// TIA Portal V20 export
FUNCTION_BLOCK "CC_Main"   // FB100, LAD
{ S7_Optimized_Access := 'TRUE' }
// stored: AutoNumber false, MemoryReserve 100, SetENOAutomatically false
   VAR_INPUT
      HMI_Reset : Bool;
      ST23_Selected : Bool;
      CNT_DownPos1 : Bool;
      CNT_DownPos2 : Bool;
      CNT_UpPos1 : Bool;
      CNT_UpPos2 : Bool;
      Hydraulic_Roller_DownPos1 : Bool;
      Hydraulic_Roller_DownPos2 : Bool;
      Hydraulic_Roller_UpPos1 : Bool;
      Hydraulic_Roller_UpPos2 : Bool;
      Drive_Roller_DownPos1 : Bool;
      Drive_Roller_DownPos2 : Bool;
      Drive_Roller_UpPos1 : Bool;
      Drive_Roller_UpPos2 : Bool;
      Module_DownPos1 : Bool;
      Module_DownPos2 : Bool;
      Module_UpPos1 : Bool;
      Module_UpPos2 : Bool;
   END_VAR
   VAR_OUTPUT
      Hydraulic_Main_Valve_Control : Bool;
   END_VAR
   VAR
      Hydraulic_Unit_Active : Bool;
      Any_Valve_Active : Bool;
      HydUnitTimerOff { S7_SetPoint := 'True'} : TON_TIME;
      HydraulicUnit_MC_Power { S7_SetPoint := 'True'} : MC_POWER;
      HydraulicUnit_MC_MoveJog { S7_SetPoint := 'True'} : MC_MOVEJOG;
      HydraulicUnit_MC_Reset { S7_SetPoint := 'True'} : MC_RESET;
      Vibrator_Control_MOD1 { S7_SetPoint := 'True'} : "CC_Vibrator_Control";
      Vibrator_Control_MOD2 { S7_SetPoint := 'True'} : "CC_Vibrator_Control";
      Vibrator_Control_MOD3 { S7_SetPoint := 'True'} : "CC_Vibrator_Control";
      Module_Control_ST23 { S7_SetPoint := 'True'} : "CC_Vib_Modules";
      ST23_UP_whenMoving { S7_SetPoint := 'True'} : Bool;
      ST24_UP_whenMoving : Bool;
      ST25_UP_whenMoving : Bool;
      MC_Power_Vib1 { S7_SetPoint := 'True'} : MC_POWER;
      MC_RESET_Vib1 { S7_SetPoint := 'True'} : MC_RESET;
      MC_MOVEJOG_Vib1 { S7_SetPoint := 'True'} : MC_MOVEJOG;
      ST24_DriveRollsUP { S7_SetPoint := 'True'} : Bool;
      ST24_DriveRollsDown : Bool;
      ST25_DriveRollsUp : Bool;
      ST25_DriveRollsDown : Bool;
      ST23_Station_Control { S7_SetPoint := 'True'} : "CC_Station_Control";
      ST24_Station_Control { S7_SetPoint := 'True'} : "CC_Station_Control";
      ST25_Station_Control { S7_SetPoint := 'True'} : "CC_Station_Control";
      ST24_Selected : Bool;
   END_VAR
   VAR CONSTANT
      STEP_RETRACT : Int := 1;
      STEP_MOVING : Int := 2;
      STEP_EXTEND : Int := 3;
   END_VAR
BEGIN

REGION Network 1
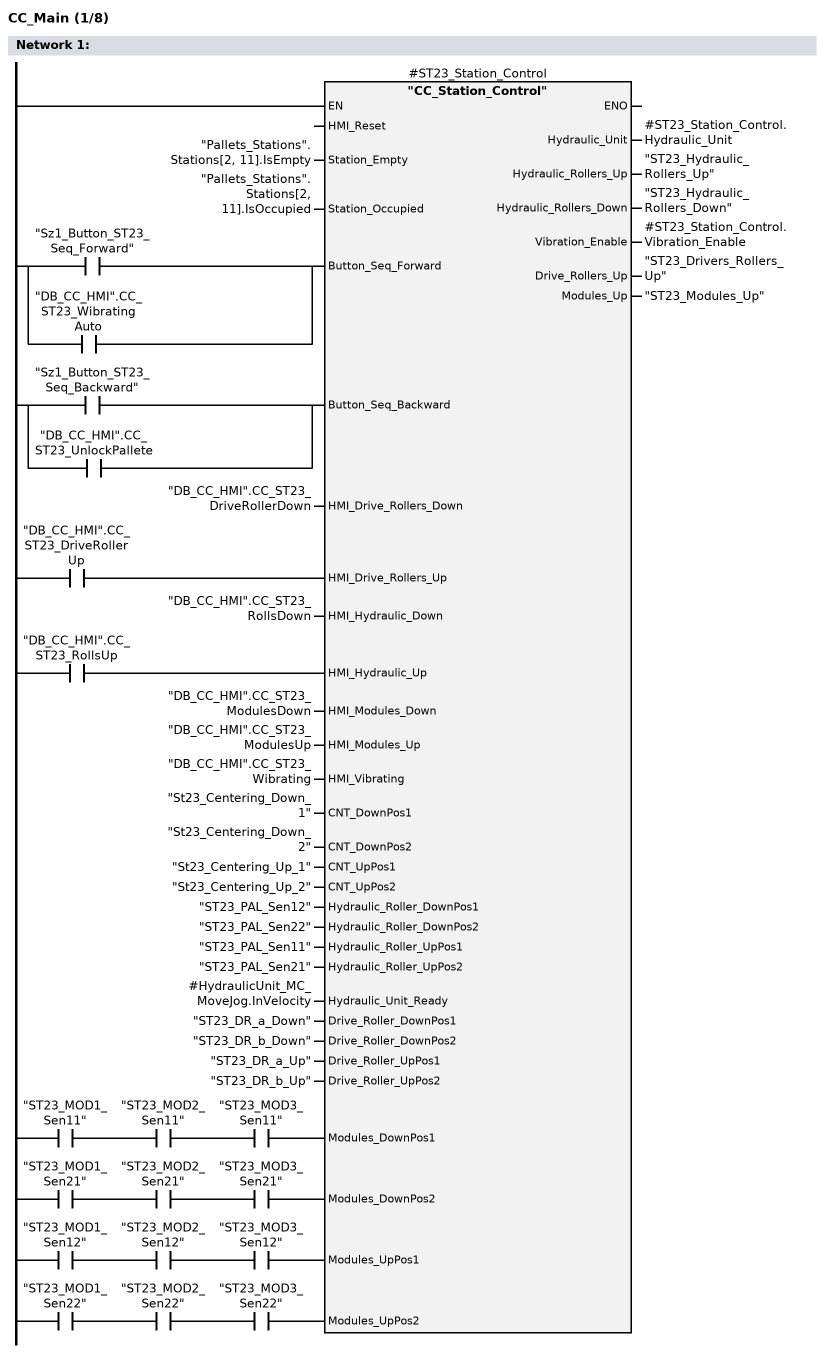
   RUNG wire#powerrail
      #ST23_Station_Control(Button_Seq_Forward := wire#w1, Button_Seq_Backward := wire#w2, HMI_Drive_Rollers_Up := wire#w3, HMI_Hydraulic_Up := wire#w4, Modules_DownPos1 := wire#w5, Modules_DownPos2 := wire#w6, Modules_UpPos1 := wire#w7, Modules_UpPos2 := wire#w8, HMI_Reset :=, Station_Empty := "Pallets_Stations".Stations[2, 11].IsEmpty, Station_Occupied := "Pallets_Stations".Stations[2, 11].IsOccupied, HMI_Drive_Rollers_Down := "DB_CC_HMI".CC_ST23_DriveRollerDown, HMI_Hydraulic_Down := "DB_CC_HMI".CC_ST23_RollsDown, HMI_Modules_Down := "DB_CC_HMI".CC_ST23_ModulesDown, HMI_Modules_Up := "DB_CC_HMI".CC_ST23_ModulesUp, HMI_Vibrating := "DB_CC_HMI".CC_ST23_Wibrating, CNT_DownPos1 := "St23_Centering_Down_1", CNT_DownPos2 := "St23_Centering_Down_2", CNT_UpPos1 := "St23_Centering_Up_1", CNT_UpPos2 := "St23_Centering_Up_2", Hydraulic_Roller_DownPos1 := "ST23_PAL_Sen12", Hydraulic_Roller_DownPos2 := "ST23_PAL_Sen22", Hydraulic_Roller_UpPos1 := "ST23_PAL_Sen11", Hydraulic_Roller_UpPos2 := "ST23_PAL_Sen21", Hydraulic_Unit_Ready := #HydraulicUnit_MC_MoveJog.InVelocity, Drive_Roller_DownPos1 := "ST23_DR_a_Down", Drive_Roller_DownPos2 := "ST23_DR_b_Down", Drive_Roller_UpPos1 := "ST23_DR_a_Up", Drive_Roller_UpPos2 := "ST23_DR_b_Up", Hydraulic_Unit => #ST23_Station_Control.Hydraulic_Unit, Hydraulic_Rollers_Up => "ST23_Hydraulic_Rollers_Up", Hydraulic_Rollers_Down => "ST23_Hydraulic_Rollers_Down", Vibration_Enable => #ST23_Station_Control.Vibration_Enable, Drive_Rollers_Up => "ST23_Drivers_Rollers_Up", Modules_Up => "ST23_Modules_Up")
   END_RUNG
   RUNG wire#powerrail
      Contact( "Sz1_Button_ST23_Seq_Forward" )
   END_RUNG wire#w1
   RUNG wire#powerrail
      Contact( "DB_CC_HMI".CC_ST23_WibratingAuto )
   END_RUNG wire#w1
   RUNG wire#powerrail
      Contact( "Sz1_Button_ST23_Seq_Backward" )
   END_RUNG wire#w2
   RUNG wire#powerrail
      Contact( "DB_CC_HMI".CC_ST23_UnlockPallete )
   END_RUNG wire#w2
   RUNG wire#powerrail
      Contact( "DB_CC_HMI".CC_ST23_DriveRollerUp )
   END_RUNG wire#w3
   RUNG wire#powerrail
      Contact( "DB_CC_HMI".CC_ST23_RollsUp )
   END_RUNG wire#w4
   RUNG wire#powerrail
      Contact( "ST23_MOD1_Sen11" )
      Contact( "ST23_MOD2_Sen11" )
      Contact( "ST23_MOD3_Sen11" )
   END_RUNG wire#w5
   RUNG wire#powerrail
      Contact( "ST23_MOD1_Sen21" )
      Contact( "ST23_MOD2_Sen21" )
      Contact( "ST23_MOD3_Sen21" )
   END_RUNG wire#w6
   RUNG wire#powerrail
      Contact( "ST23_MOD1_Sen12" )
      Contact( "ST23_MOD2_Sen12" )
      Contact( "ST23_MOD3_Sen12" )
   END_RUNG wire#w7
   RUNG wire#powerrail
      Contact( "ST23_MOD1_Sen22" )
      Contact( "ST23_MOD2_Sen22" )
      Contact( "ST23_MOD3_Sen22" )
   END_RUNG wire#w8
   // the same network as SCL:
   #ST23_Station_Control(Station_Empty := "Pallets_Stations".Stations[2, 11].IsEmpty,   // "CC_Station_Control"
                         Station_Occupied := "Pallets_Stations".Stations[2, 11].IsOccupied,
                         Button_Seq_Forward := "Sz1_Button_ST23_Seq_Forward" OR "DB_CC_HMI".CC_ST23_WibratingAuto,
                         Button_Seq_Backward := "Sz1_Button_ST23_Seq_Backward" OR "DB_CC_HMI".CC_ST23_UnlockPallete,
                         HMI_Drive_Rollers_Down := "DB_CC_HMI".CC_ST23_DriveRollerDown,
                         HMI_Drive_Rollers_Up := "DB_CC_HMI".CC_ST23_DriveRollerUp,
                         HMI_Hydraulic_Down := "DB_CC_HMI".CC_ST23_RollsDown,
                         HMI_Hydraulic_Up := "DB_CC_HMI".CC_ST23_RollsUp,
                         HMI_Modules_Down := "DB_CC_HMI".CC_ST23_ModulesDown,
                         HMI_Modules_Up := "DB_CC_HMI".CC_ST23_ModulesUp,
                         HMI_Vibrating := "DB_CC_HMI".CC_ST23_Wibrating,
                         CNT_DownPos1 := "St23_Centering_Down_1",
                         CNT_DownPos2 := "St23_Centering_Down_2",
                         CNT_UpPos1 := "St23_Centering_Up_1",
                         CNT_UpPos2 := "St23_Centering_Up_2",
                         Hydraulic_Roller_DownPos1 := "ST23_PAL_Sen12",
                         Hydraulic_Roller_DownPos2 := "ST23_PAL_Sen22",
                         Hydraulic_Roller_UpPos1 := "ST23_PAL_Sen11",
                         Hydraulic_Roller_UpPos2 := "ST23_PAL_Sen21",
                         Hydraulic_Unit_Ready := #HydraulicUnit_MC_MoveJog.InVelocity,
                         Drive_Roller_DownPos1 := "ST23_DR_a_Down",
                         Drive_Roller_DownPos2 := "ST23_DR_b_Down",
                         Drive_Roller_UpPos1 := "ST23_DR_a_Up",
                         Drive_Roller_UpPos2 := "ST23_DR_b_Up",
                         Modules_DownPos1 := "ST23_MOD1_Sen11" AND "ST23_MOD2_Sen11" AND "ST23_MOD3_Sen11",
                         Modules_DownPos2 := "ST23_MOD1_Sen21" AND "ST23_MOD2_Sen21" AND "ST23_MOD3_Sen21",
                         Modules_UpPos1 := "ST23_MOD1_Sen12" AND "ST23_MOD2_Sen12" AND "ST23_MOD3_Sen12",
                         Modules_UpPos2 := "ST23_MOD1_Sen22" AND "ST23_MOD2_Sen22" AND "ST23_MOD3_Sen22",
                         Hydraulic_Unit => #ST23_Station_Control.Hydraulic_Unit,
                         Hydraulic_Rollers_Up => "ST23_Hydraulic_Rollers_Up",
                         Hydraulic_Rollers_Down => "ST23_Hydraulic_Rollers_Down",
                         Vibration_Enable => #ST23_Station_Control.Vibration_Enable,
                         Drive_Rollers_Up => "ST23_Drivers_Rollers_Up",
                         Modules_Up => "ST23_Modules_Up");
END_REGION

REGION Network 2
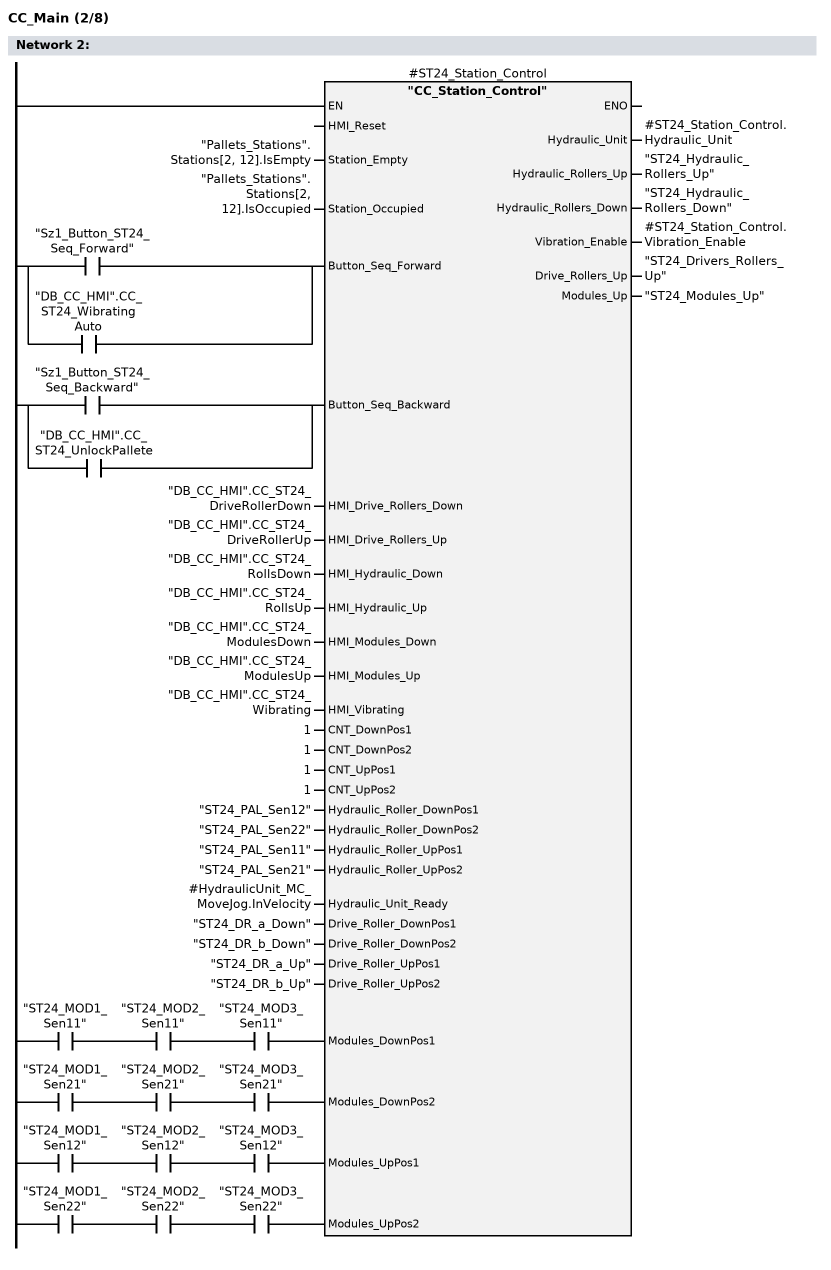
   RUNG wire#powerrail
      #ST24_Station_Control(Button_Seq_Forward := wire#w1, Button_Seq_Backward := wire#w2, Modules_DownPos1 := wire#w3, Modules_DownPos2 := wire#w4, Modules_UpPos1 := wire#w5, Modules_UpPos2 := wire#w6, HMI_Reset :=, Station_Empty := "Pallets_Stations".Stations[2, 12].IsEmpty, Station_Occupied := "Pallets_Stations".Stations[2, 12].IsOccupied, HMI_Drive_Rollers_Down := "DB_CC_HMI".CC_ST24_DriveRollerDown, HMI_Drive_Rollers_Up := "DB_CC_HMI".CC_ST24_DriveRollerUp, HMI_Hydraulic_Down := "DB_CC_HMI".CC_ST24_RollsDown, HMI_Hydraulic_Up := "DB_CC_HMI".CC_ST24_RollsUp, HMI_Modules_Down := "DB_CC_HMI".CC_ST24_ModulesDown, HMI_Modules_Up := "DB_CC_HMI".CC_ST24_ModulesUp, HMI_Vibrating := "DB_CC_HMI".CC_ST24_Wibrating, CNT_DownPos1 := 1, CNT_DownPos2 := 1, CNT_UpPos1 := 1, CNT_UpPos2 := 1, Hydraulic_Roller_DownPos1 := "ST24_PAL_Sen12", Hydraulic_Roller_DownPos2 := "ST24_PAL_Sen22", Hydraulic_Roller_UpPos1 := "ST24_PAL_Sen11", Hydraulic_Roller_UpPos2 := "ST24_PAL_Sen21", Hydraulic_Unit_Ready := #HydraulicUnit_MC_MoveJog.InVelocity, Drive_Roller_DownPos1 := "ST24_DR_a_Down", Drive_Roller_DownPos2 := "ST24_DR_b_Down", Drive_Roller_UpPos1 := "ST24_DR_a_Up", Drive_Roller_UpPos2 := "ST24_DR_b_Up", Hydraulic_Unit => #ST24_Station_Control.Hydraulic_Unit, Hydraulic_Rollers_Up => "ST24_Hydraulic_Rollers_Up", Hydraulic_Rollers_Down => "ST24_Hydraulic_Rollers_Down", Vibration_Enable => #ST24_Station_Control.Vibration_Enable, Drive_Rollers_Up => "ST24_Drivers_Rollers_Up", Modules_Up => "ST24_Modules_Up")
   END_RUNG
   RUNG wire#powerrail
      Contact( "Sz1_Button_ST24_Seq_Forward" )
   END_RUNG wire#w1
   RUNG wire#powerrail
      Contact( "DB_CC_HMI".CC_ST24_WibratingAuto )
   END_RUNG wire#w1
   RUNG wire#powerrail
      Contact( "Sz1_Button_ST24_Seq_Backward" )
   END_RUNG wire#w2
   RUNG wire#powerrail
      Contact( "DB_CC_HMI".CC_ST24_UnlockPallete )
   END_RUNG wire#w2
   RUNG wire#powerrail
      Contact( "ST24_MOD1_Sen11" )
      Contact( "ST24_MOD2_Sen11" )
      Contact( "ST24_MOD3_Sen11" )
   END_RUNG wire#w3
   RUNG wire#powerrail
      Contact( "ST24_MOD1_Sen21" )
      Contact( "ST24_MOD2_Sen21" )
      Contact( "ST24_MOD3_Sen21" )
   END_RUNG wire#w4
   RUNG wire#powerrail
      Contact( "ST24_MOD1_Sen12" )
      Contact( "ST24_MOD2_Sen12" )
      Contact( "ST24_MOD3_Sen12" )
   END_RUNG wire#w5
   RUNG wire#powerrail
      Contact( "ST24_MOD1_Sen22" )
      Contact( "ST24_MOD2_Sen22" )
      Contact( "ST24_MOD3_Sen22" )
   END_RUNG wire#w6
   // the same network as SCL:
   #ST24_Station_Control(Station_Empty := "Pallets_Stations".Stations[2, 12].IsEmpty,   // "CC_Station_Control"
                         Station_Occupied := "Pallets_Stations".Stations[2, 12].IsOccupied,
                         Button_Seq_Forward := "Sz1_Button_ST24_Seq_Forward" OR "DB_CC_HMI".CC_ST24_WibratingAuto,
                         Button_Seq_Backward := "Sz1_Button_ST24_Seq_Backward" OR "DB_CC_HMI".CC_ST24_UnlockPallete,
                         HMI_Drive_Rollers_Down := "DB_CC_HMI".CC_ST24_DriveRollerDown,
                         HMI_Drive_Rollers_Up := "DB_CC_HMI".CC_ST24_DriveRollerUp,
                         HMI_Hydraulic_Down := "DB_CC_HMI".CC_ST24_RollsDown,
                         HMI_Hydraulic_Up := "DB_CC_HMI".CC_ST24_RollsUp,
                         HMI_Modules_Down := "DB_CC_HMI".CC_ST24_ModulesDown,
                         HMI_Modules_Up := "DB_CC_HMI".CC_ST24_ModulesUp,
                         HMI_Vibrating := "DB_CC_HMI".CC_ST24_Wibrating,
                         CNT_DownPos1 := 1,
                         CNT_DownPos2 := 1,
                         CNT_UpPos1 := 1,
                         CNT_UpPos2 := 1,
                         Hydraulic_Roller_DownPos1 := "ST24_PAL_Sen12",
                         Hydraulic_Roller_DownPos2 := "ST24_PAL_Sen22",
                         Hydraulic_Roller_UpPos1 := "ST24_PAL_Sen11",
                         Hydraulic_Roller_UpPos2 := "ST24_PAL_Sen21",
                         Hydraulic_Unit_Ready := #HydraulicUnit_MC_MoveJog.InVelocity,
                         Drive_Roller_DownPos1 := "ST24_DR_a_Down",
                         Drive_Roller_DownPos2 := "ST24_DR_b_Down",
                         Drive_Roller_UpPos1 := "ST24_DR_a_Up",
                         Drive_Roller_UpPos2 := "ST24_DR_b_Up",
                         Modules_DownPos1 := "ST24_MOD1_Sen11" AND "ST24_MOD2_Sen11" AND "ST24_MOD3_Sen11",
                         Modules_DownPos2 := "ST24_MOD1_Sen21" AND "ST24_MOD2_Sen21" AND "ST24_MOD3_Sen21",
                         Modules_UpPos1 := "ST24_MOD1_Sen12" AND "ST24_MOD2_Sen12" AND "ST24_MOD3_Sen12",
                         Modules_UpPos2 := "ST24_MOD1_Sen22" AND "ST24_MOD2_Sen22" AND "ST24_MOD3_Sen22",
                         Hydraulic_Unit => #ST24_Station_Control.Hydraulic_Unit,
                         Hydraulic_Rollers_Up => "ST24_Hydraulic_Rollers_Up",
                         Hydraulic_Rollers_Down => "ST24_Hydraulic_Rollers_Down",
                         Vibration_Enable => #ST24_Station_Control.Vibration_Enable,
                         Drive_Rollers_Up => "ST24_Drivers_Rollers_Up",
                         Modules_Up => "ST24_Modules_Up");
END_REGION

REGION Network 3
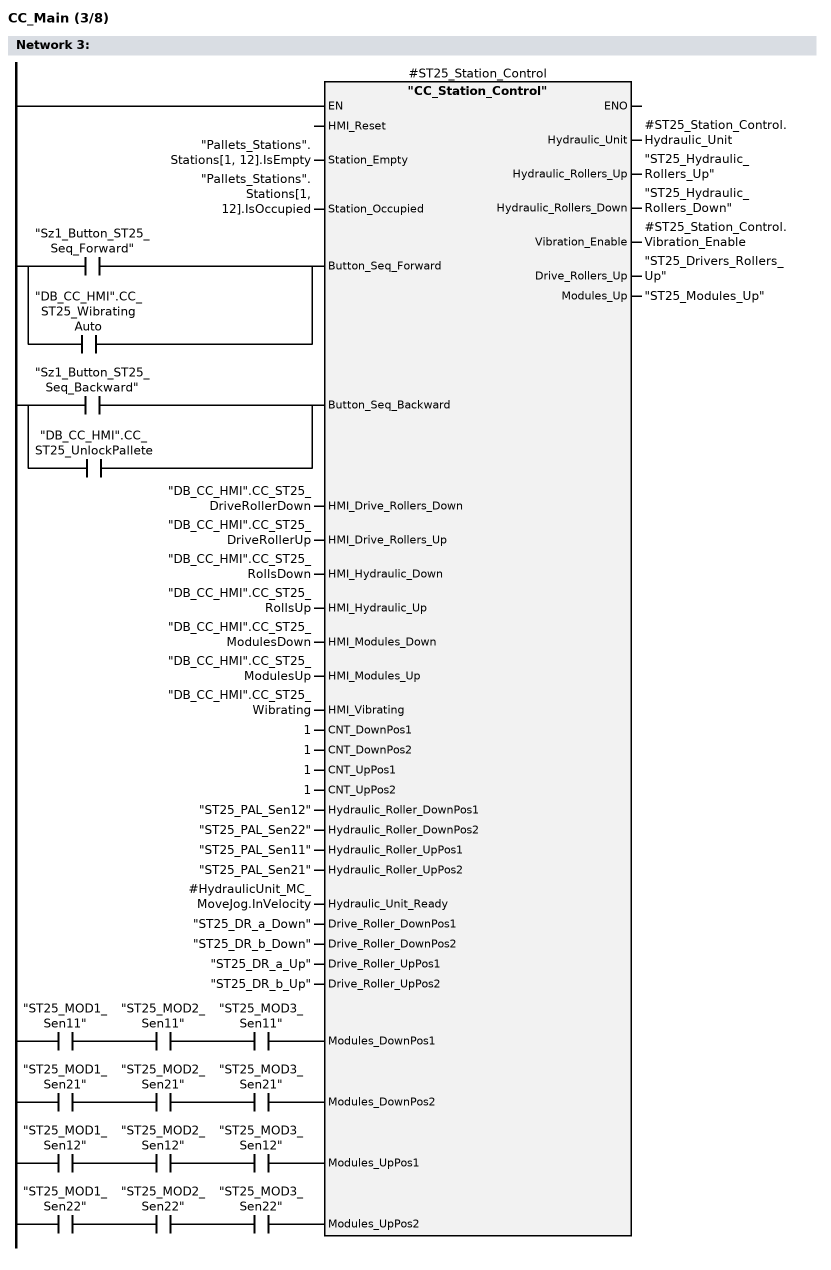
   RUNG wire#powerrail
      #ST25_Station_Control(Button_Seq_Forward := wire#w1, Button_Seq_Backward := wire#w2, Modules_DownPos1 := wire#w3, Modules_DownPos2 := wire#w4, Modules_UpPos1 := wire#w5, Modules_UpPos2 := wire#w6, HMI_Reset :=, Station_Empty := "Pallets_Stations".Stations[1, 12].IsEmpty, Station_Occupied := "Pallets_Stations".Stations[1, 12].IsOccupied, HMI_Drive_Rollers_Down := "DB_CC_HMI".CC_ST25_DriveRollerDown, HMI_Drive_Rollers_Up := "DB_CC_HMI".CC_ST25_DriveRollerUp, HMI_Hydraulic_Down := "DB_CC_HMI".CC_ST25_RollsDown, HMI_Hydraulic_Up := "DB_CC_HMI".CC_ST25_RollsUp, HMI_Modules_Down := "DB_CC_HMI".CC_ST25_ModulesDown, HMI_Modules_Up := "DB_CC_HMI".CC_ST25_ModulesUp, HMI_Vibrating := "DB_CC_HMI".CC_ST25_Wibrating, CNT_DownPos1 := 1, CNT_DownPos2 := 1, CNT_UpPos1 := 1, CNT_UpPos2 := 1, Hydraulic_Roller_DownPos1 := "ST25_PAL_Sen12", Hydraulic_Roller_DownPos2 := "ST25_PAL_Sen22", Hydraulic_Roller_UpPos1 := "ST25_PAL_Sen11", Hydraulic_Roller_UpPos2 := "ST25_PAL_Sen21", Hydraulic_Unit_Ready := #HydraulicUnit_MC_MoveJog.InVelocity, Drive_Roller_DownPos1 := "ST25_DR_a_Down", Drive_Roller_DownPos2 := "ST25_DR_b_Down", Drive_Roller_UpPos1 := "ST25_DR_a_Up", Drive_Roller_UpPos2 := "ST25_DR_b_Up", Hydraulic_Unit => #ST25_Station_Control.Hydraulic_Unit, Hydraulic_Rollers_Up => "ST25_Hydraulic_Rollers_Up", Hydraulic_Rollers_Down => "ST25_Hydraulic_Rollers_Down", Vibration_Enable => #ST25_Station_Control.Vibration_Enable, Drive_Rollers_Up => "ST25_Drivers_Rollers_Up", Modules_Up => "ST25_Modules_Up")
   END_RUNG
   RUNG wire#powerrail
      Contact( "Sz1_Button_ST25_Seq_Forward" )
   END_RUNG wire#w1
   RUNG wire#powerrail
      Contact( "DB_CC_HMI".CC_ST25_WibratingAuto )
   END_RUNG wire#w1
   RUNG wire#powerrail
      Contact( "Sz1_Button_ST25_Seq_Backward" )
   END_RUNG wire#w2
   RUNG wire#powerrail
      Contact( "DB_CC_HMI".CC_ST25_UnlockPallete )
   END_RUNG wire#w2
   RUNG wire#powerrail
      Contact( "ST25_MOD1_Sen11" )
      Contact( "ST25_MOD2_Sen11" )
      Contact( "ST25_MOD3_Sen11" )
   END_RUNG wire#w3
   RUNG wire#powerrail
      Contact( "ST25_MOD1_Sen21" )
      Contact( "ST25_MOD2_Sen21" )
      Contact( "ST25_MOD3_Sen21" )
   END_RUNG wire#w4
   RUNG wire#powerrail
      Contact( "ST25_MOD1_Sen12" )
      Contact( "ST25_MOD2_Sen12" )
      Contact( "ST25_MOD3_Sen12" )
   END_RUNG wire#w5
   RUNG wire#powerrail
      Contact( "ST25_MOD1_Sen22" )
      Contact( "ST25_MOD2_Sen22" )
      Contact( "ST25_MOD3_Sen22" )
   END_RUNG wire#w6
   // the same network as SCL:
   #ST25_Station_Control(Station_Empty := "Pallets_Stations".Stations[1, 12].IsEmpty,   // "CC_Station_Control"
                         Station_Occupied := "Pallets_Stations".Stations[1, 12].IsOccupied,
                         Button_Seq_Forward := "Sz1_Button_ST25_Seq_Forward" OR "DB_CC_HMI".CC_ST25_WibratingAuto,
                         Button_Seq_Backward := "Sz1_Button_ST25_Seq_Backward" OR "DB_CC_HMI".CC_ST25_UnlockPallete,
                         HMI_Drive_Rollers_Down := "DB_CC_HMI".CC_ST25_DriveRollerDown,
                         HMI_Drive_Rollers_Up := "DB_CC_HMI".CC_ST25_DriveRollerUp,
                         HMI_Hydraulic_Down := "DB_CC_HMI".CC_ST25_RollsDown,
                         HMI_Hydraulic_Up := "DB_CC_HMI".CC_ST25_RollsUp,
                         HMI_Modules_Down := "DB_CC_HMI".CC_ST25_ModulesDown,
                         HMI_Modules_Up := "DB_CC_HMI".CC_ST25_ModulesUp,
                         HMI_Vibrating := "DB_CC_HMI".CC_ST25_Wibrating,
                         CNT_DownPos1 := 1,
                         CNT_DownPos2 := 1,
                         CNT_UpPos1 := 1,
                         CNT_UpPos2 := 1,
                         Hydraulic_Roller_DownPos1 := "ST25_PAL_Sen12",
                         Hydraulic_Roller_DownPos2 := "ST25_PAL_Sen22",
                         Hydraulic_Roller_UpPos1 := "ST25_PAL_Sen11",
                         Hydraulic_Roller_UpPos2 := "ST25_PAL_Sen21",
                         Hydraulic_Unit_Ready := #HydraulicUnit_MC_MoveJog.InVelocity,
                         Drive_Roller_DownPos1 := "ST25_DR_a_Down",
                         Drive_Roller_DownPos2 := "ST25_DR_b_Down",
                         Drive_Roller_UpPos1 := "ST25_DR_a_Up",
                         Drive_Roller_UpPos2 := "ST25_DR_b_Up",
                         Modules_DownPos1 := "ST25_MOD1_Sen11" AND "ST25_MOD2_Sen11" AND "ST25_MOD3_Sen11",
                         Modules_DownPos2 := "ST25_MOD1_Sen21" AND "ST25_MOD2_Sen21" AND "ST25_MOD3_Sen21",
                         Modules_UpPos1 := "ST25_MOD1_Sen12" AND "ST25_MOD2_Sen12" AND "ST25_MOD3_Sen12",
                         Modules_UpPos2 := "ST25_MOD1_Sen22" AND "ST25_MOD2_Sen22" AND "ST25_MOD3_Sen22",
                         Hydraulic_Unit => #ST25_Station_Control.Hydraulic_Unit,
                         Hydraulic_Rollers_Up => "ST25_Hydraulic_Rollers_Up",
                         Hydraulic_Rollers_Down => "ST25_Hydraulic_Rollers_Down",
                         Vibration_Enable => #ST25_Station_Control.Vibration_Enable,
                         Drive_Rollers_Up => "ST25_Drivers_Rollers_Up",
                         Modules_Up => "ST25_Modules_Up");
END_REGION

REGION Network 4: Data to safety set hydraulic main valve
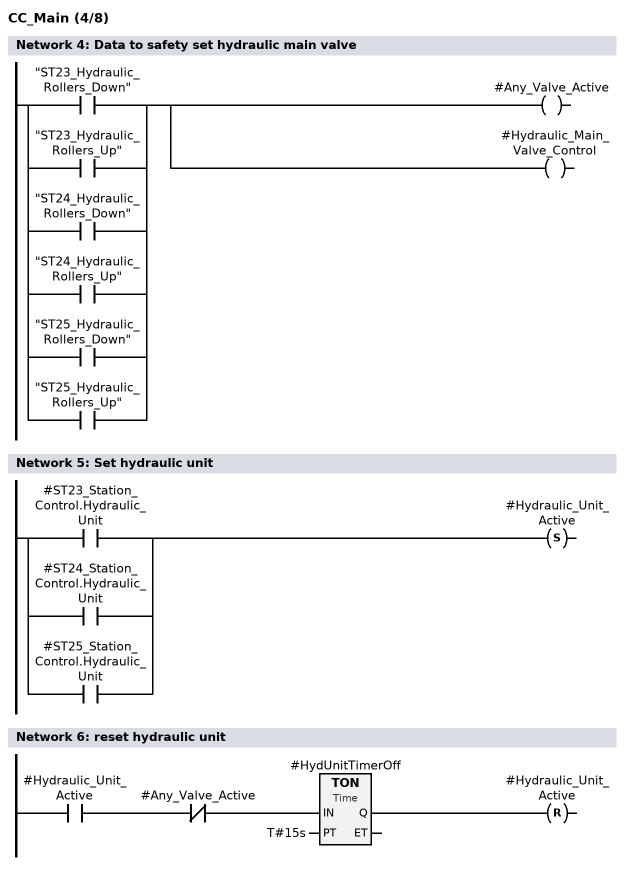
   RUNG wire#powerrail
      Contact( "ST23_Hydraulic_Rollers_Down" )
      wire#w1
      Coil( #Any_Valve_Active )
   END_RUNG
   RUNG wire#powerrail
      Contact( "ST23_Hydraulic_Rollers_Up" )
   END_RUNG wire#w1
   RUNG wire#powerrail
      Contact( "ST24_Hydraulic_Rollers_Down" )
   END_RUNG wire#w1
   RUNG wire#powerrail
      Contact( "ST24_Hydraulic_Rollers_Up" )
   END_RUNG wire#w1
   RUNG wire#powerrail
      Contact( "ST25_Hydraulic_Rollers_Down" )
   END_RUNG wire#w1
   RUNG wire#powerrail
      Contact( "ST25_Hydraulic_Rollers_Up" )
   END_RUNG wire#w1
   RUNG wire#w1
      Coil( #Hydraulic_Main_Valve_Control )
   END_RUNG
   // the same network as SCL:
   #Any_Valve_Active := "ST23_Hydraulic_Rollers_Down" OR "ST23_Hydraulic_Rollers_Up" OR "ST24_Hydraulic_Rollers_Down" OR "ST24_Hydraulic_Rollers_Up" OR "ST25_Hydraulic_Rollers_Down" OR "ST25_Hydraulic_Rollers_Up";
   #Hydraulic_Main_Valve_Control := #Any_Valve_Active;
END_REGION

REGION Network 5: Set hydraulic unit
   RUNG wire#powerrail
      Contact( #ST23_Station_Control.Hydraulic_Unit )
      wire#w1
      S_Coil( #Hydraulic_Unit_Active )
   END_RUNG
   RUNG wire#powerrail
      Contact( #ST24_Station_Control.Hydraulic_Unit )
   END_RUNG wire#w1
   RUNG wire#powerrail
      Contact( #ST25_Station_Control.Hydraulic_Unit )
   END_RUNG wire#w1
   // the same network as SCL:
   IF #ST23_Station_Control.Hydraulic_Unit OR #ST24_Station_Control.Hydraulic_Unit OR #ST25_Station_Control.Hydraulic_Unit THEN
       #Hydraulic_Unit_Active := TRUE;
   END_IF;
END_REGION

REGION Network 6: reset hydraulic unit
   RUNG wire#powerrail
      Contact( #Hydraulic_Unit_Active )
      I_Contact( #Any_Valve_Active )
      { S7_Templates := "time_type := Time" } #HydUnitTimerOff.TON(pt := T#15s, et =>)
      R_Coil( #Hydraulic_Unit_Active )
   END_RUNG
   // the same network as SCL:
   #HydUnitTimerOff(IN := #Hydraulic_Unit_Active AND NOT #Any_Valve_Active, PT := T#15s);   // TON
   IF #HydUnitTimerOff.Q THEN #Hydraulic_Unit_Active := FALSE; END_IF;
END_REGION

REGION Network 7: Hydraulic Unit Motion Control
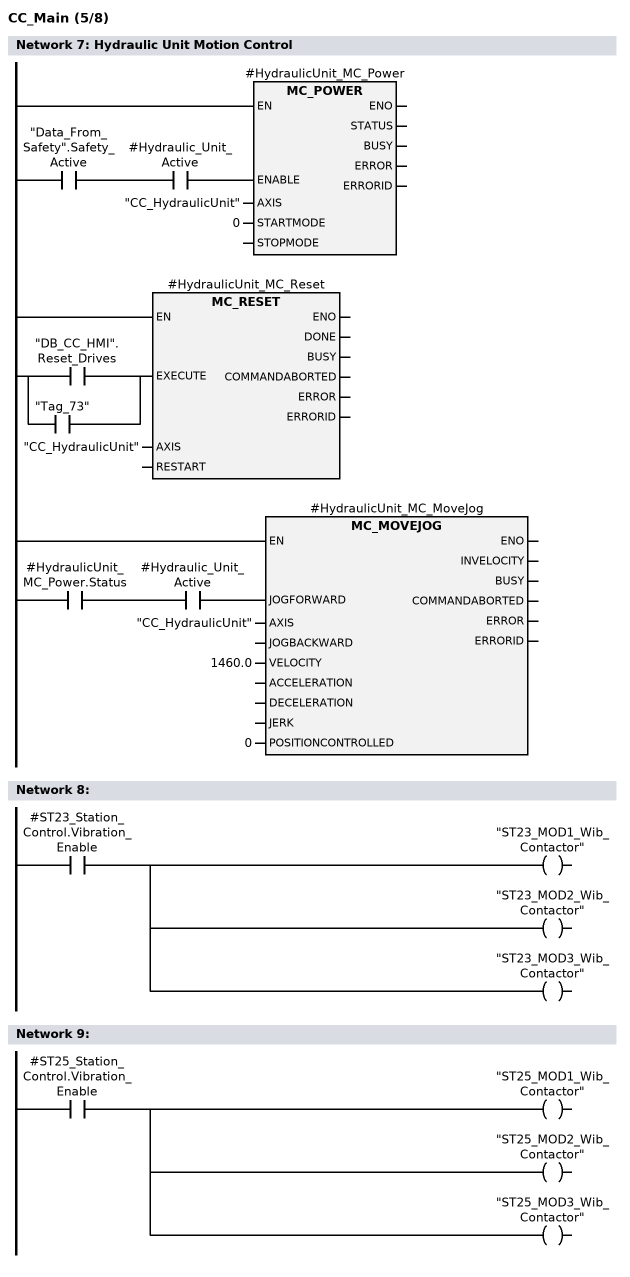
   RUNG wire#powerrail
      #HydraulicUnit_MC_Power.MC_POWER(Enable := wire#w1, Axis := "CC_HydraulicUnit", StartMode := 0, StopMode :=, Status =>, Busy =>, Error =>, ErrorId =>)
   END_RUNG
   RUNG wire#powerrail
      Contact( "Data_From_Safety".Safety_Active )
      Contact( #Hydraulic_Unit_Active )
   END_RUNG wire#w1
   RUNG wire#powerrail
      #HydraulicUnit_MC_Reset.MC_RESET(Execute := wire#w2, Axis := "CC_HydraulicUnit", Restart :=, Done =>, Busy =>, CommandAborted =>, Error =>, ErrorId =>)
   END_RUNG
   RUNG wire#powerrail
      Contact( "DB_CC_HMI".Reset_Drives )
   END_RUNG wire#w2
   RUNG wire#powerrail
      Contact( "Tag_73" )
   END_RUNG wire#w2
   RUNG wire#powerrail
      #HydraulicUnit_MC_MoveJog.MC_MOVEJOG(JogForward := wire#w3, Axis := "CC_HydraulicUnit", JogBackward :=, Velocity := 1460.0, Acceleration :=, Deceleration :=, Jerk :=, PositionControlled := 0, InVelocity =>, Busy =>, CommandAborted =>, Error =>, ErrorId =>)
   END_RUNG
   RUNG wire#powerrail
      Contact( #HydraulicUnit_MC_Power.Status )
      Contact( #Hydraulic_Unit_Active )
   END_RUNG wire#w3
   // the same network as SCL:
   #HydraulicUnit_MC_Power(Enable := "Data_From_Safety".Safety_Active AND #Hydraulic_Unit_Active,   // MC_POWER
                           Axis := "CC_HydraulicUnit",
                           StartMode := 0);
   #HydraulicUnit_MC_Reset(Execute := "DB_CC_HMI".Reset_Drives OR "Tag_73", Axis := "CC_HydraulicUnit");   // MC_RESET
   #HydraulicUnit_MC_MoveJog(JogForward := #HydraulicUnit_MC_Power.Status AND #Hydraulic_Unit_Active,   // MC_MOVEJOG
                           Axis := "CC_HydraulicUnit",
                           Velocity := 1460.0,
                           PositionControlled := 0);
END_REGION

REGION Network 8
   RUNG wire#powerrail
      Contact( #ST23_Station_Control.Vibration_Enable )
      wire#w1
      Coil( "ST23_MOD1_Wib_Contactor" )
   END_RUNG
   RUNG wire#w1
      Coil( "ST23_MOD2_Wib_Contactor" )
   END_RUNG
   RUNG wire#w1
      Coil( "ST23_MOD3_Wib_Contactor" )
   END_RUNG
   // the same network as SCL:
   "ST23_MOD1_Wib_Contactor" := #ST23_Station_Control.Vibration_Enable;
   "ST23_MOD2_Wib_Contactor" := #ST23_Station_Control.Vibration_Enable;
   "ST23_MOD3_Wib_Contactor" := #ST23_Station_Control.Vibration_Enable;
END_REGION

REGION Network 9
   RUNG wire#powerrail
      Contact( #ST25_Station_Control.Vibration_Enable )
      wire#w1
      Coil( "ST25_MOD1_Wib_Contactor" )
   END_RUNG
   RUNG wire#w1
      Coil( "ST25_MOD2_Wib_Contactor" )
   END_RUNG
   RUNG wire#w1
      Coil( "ST25_MOD3_Wib_Contactor" )
   END_RUNG
   // the same network as SCL:
   "ST25_MOD1_Wib_Contactor" := #ST25_Station_Control.Vibration_Enable;
   "ST25_MOD2_Wib_Contactor" := #ST25_Station_Control.Vibration_Enable;
   "ST25_MOD3_Wib_Contactor" := #ST25_Station_Control.Vibration_Enable;
END_REGION

REGION Network 10
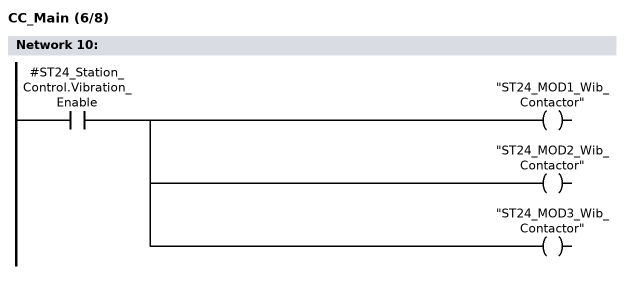
   RUNG wire#powerrail
      Contact( #ST24_Station_Control.Vibration_Enable )
      wire#w1
      Coil( "ST24_MOD1_Wib_Contactor" )
   END_RUNG
   RUNG wire#w1
      Coil( "ST24_MOD2_Wib_Contactor" )
   END_RUNG
   RUNG wire#w1
      Coil( "ST24_MOD3_Wib_Contactor" )
   END_RUNG
   // the same network as SCL:
   "ST24_MOD1_Wib_Contactor" := #ST24_Station_Control.Vibration_Enable;
   "ST24_MOD2_Wib_Contactor" := #ST24_Station_Control.Vibration_Enable;
   "ST24_MOD3_Wib_Contactor" := #ST24_Station_Control.Vibration_Enable;
END_REGION

REGION Network 11
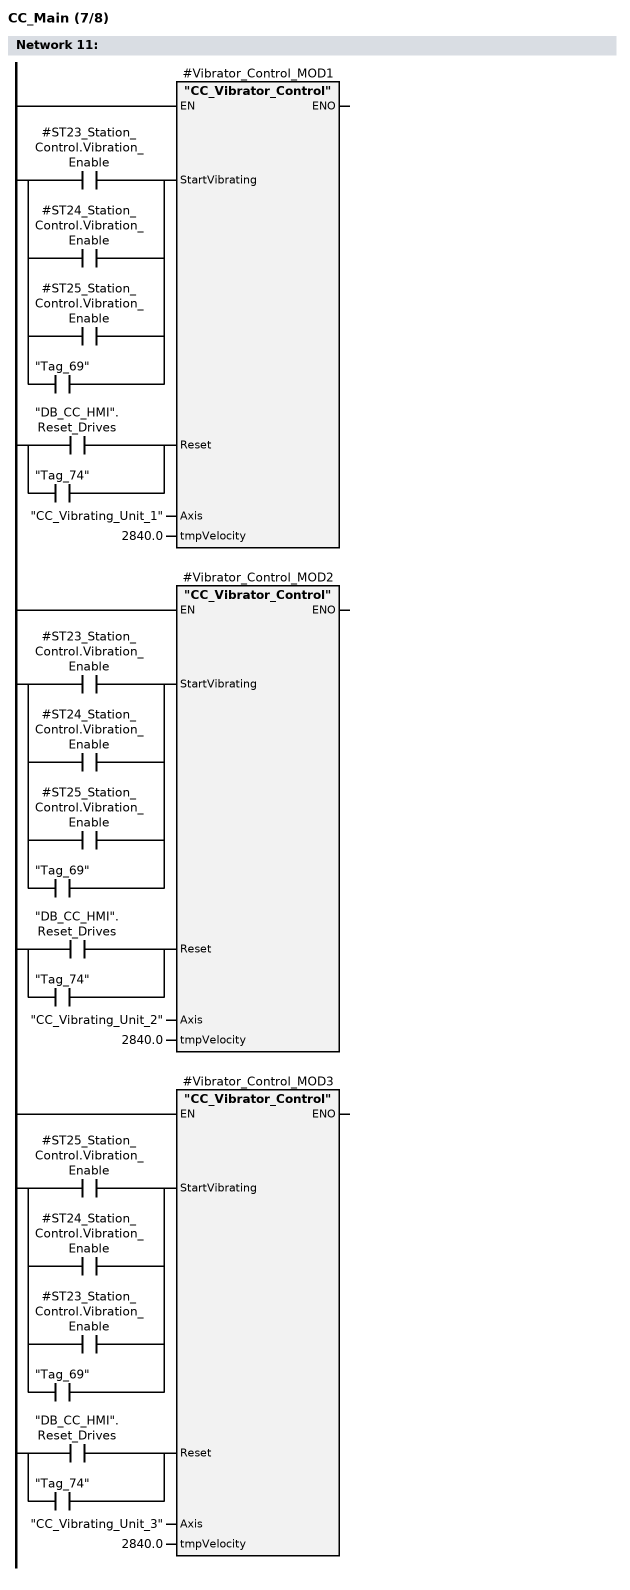
   RUNG wire#powerrail
      #Vibrator_Control_MOD1(StartVibrating := wire#w1, Reset := wire#w2, Axis := "CC_Vibrating_Unit_1", tmpVelocity := 2840.0)
   END_RUNG
   RUNG wire#powerrail
      Contact( #ST23_Station_Control.Vibration_Enable )
   END_RUNG wire#w1
   RUNG wire#powerrail
      Contact( #ST24_Station_Control.Vibration_Enable )
   END_RUNG wire#w1
   RUNG wire#powerrail
      Contact( #ST25_Station_Control.Vibration_Enable )
   END_RUNG wire#w1
   RUNG wire#powerrail
      Contact( "Tag_69" )
   END_RUNG wire#w1
   RUNG wire#powerrail
      Contact( "DB_CC_HMI".Reset_Drives )
   END_RUNG wire#w2
   RUNG wire#powerrail
      Contact( "Tag_74" )
   END_RUNG wire#w2
   RUNG wire#powerrail
      #Vibrator_Control_MOD2(StartVibrating := wire#w3, Reset := wire#w4, Axis := "CC_Vibrating_Unit_2", tmpVelocity := 2840.0)
   END_RUNG
   RUNG wire#powerrail
      Contact( #ST23_Station_Control.Vibration_Enable )
   END_RUNG wire#w3
   RUNG wire#powerrail
      Contact( #ST24_Station_Control.Vibration_Enable )
   END_RUNG wire#w3
   RUNG wire#powerrail
      Contact( #ST25_Station_Control.Vibration_Enable )
   END_RUNG wire#w3
   RUNG wire#powerrail
      Contact( "Tag_69" )
   END_RUNG wire#w3
   RUNG wire#powerrail
      Contact( "DB_CC_HMI".Reset_Drives )
   END_RUNG wire#w4
   RUNG wire#powerrail
      Contact( "Tag_74" )
   END_RUNG wire#w4
   RUNG wire#powerrail
      #Vibrator_Control_MOD3(StartVibrating := wire#w5, Reset := wire#w6, Axis := "CC_Vibrating_Unit_3", tmpVelocity := 2840.0)
   END_RUNG
   RUNG wire#powerrail
      Contact( #ST25_Station_Control.Vibration_Enable )
   END_RUNG wire#w5
   RUNG wire#powerrail
      Contact( #ST24_Station_Control.Vibration_Enable )
   END_RUNG wire#w5
   RUNG wire#powerrail
      Contact( #ST23_Station_Control.Vibration_Enable )
   END_RUNG wire#w5
   RUNG wire#powerrail
      Contact( "Tag_69" )
   END_RUNG wire#w5
   RUNG wire#powerrail
      Contact( "DB_CC_HMI".Reset_Drives )
   END_RUNG wire#w6
   RUNG wire#powerrail
      Contact( "Tag_74" )
   END_RUNG wire#w6
   // the same network as SCL:
   #Vibrator_Control_MOD1(StartVibrating := #ST23_Station_Control.Vibration_Enable OR #ST24_Station_Control.Vibration_Enable OR #ST25_Station_Control.Vibration_Enable OR "Tag_69",   // "CC_Vibrator_Control"
                          Reset := "DB_CC_HMI".Reset_Drives OR "Tag_74",
                          Axis := "CC_Vibrating_Unit_1",
                          tmpVelocity := 2840.0);
   #Vibrator_Control_MOD2(StartVibrating := #ST23_Station_Control.Vibration_Enable OR #ST24_Station_Control.Vibration_Enable OR #ST25_Station_Control.Vibration_Enable OR "Tag_69",   // "CC_Vibrator_Control"
                          Reset := "DB_CC_HMI".Reset_Drives OR "Tag_74",
                          Axis := "CC_Vibrating_Unit_2",
                          tmpVelocity := 2840.0);
   #Vibrator_Control_MOD3(StartVibrating := #ST25_Station_Control.Vibration_Enable OR #ST24_Station_Control.Vibration_Enable OR #ST23_Station_Control.Vibration_Enable OR "Tag_69",   // "CC_Vibrator_Control"
                          Reset := "DB_CC_HMI".Reset_Drives OR "Tag_74",
                          Axis := "CC_Vibrating_Unit_3",
                          tmpVelocity := 2840.0);
END_REGION

REGION Network 12
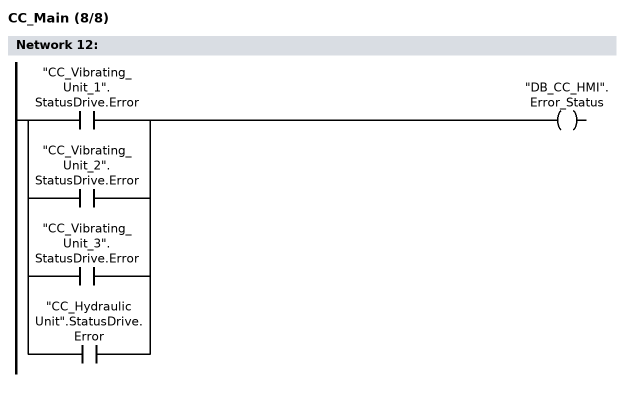
   RUNG wire#powerrail
      Contact( "CC_Vibrating_Unit_1".StatusDrive.Error )
      wire#w1
      Coil( "DB_CC_HMI".Error_Status )
   END_RUNG
   RUNG wire#powerrail
      Contact( "CC_Vibrating_Unit_2".StatusDrive.Error )
   END_RUNG wire#w1
   RUNG wire#powerrail
      Contact( "CC_Vibrating_Unit_3".StatusDrive.Error )
   END_RUNG wire#w1
   RUNG wire#powerrail
      Contact( "CC_HydraulicUnit".StatusDrive.Error )
   END_RUNG wire#w1
   // the same network as SCL:
   "DB_CC_HMI".Error_Status := "CC_Vibrating_Unit_1".StatusDrive.Error OR "CC_Vibrating_Unit_2".StatusDrive.Error OR "CC_Vibrating_Unit_3".StatusDrive.Error OR "CC_HydraulicUnit".StatusDrive.Error;
END_REGION
END_FUNCTION_BLOCK
